(* PLC project marvel_solar, Institute of Astronomy Onto 0.0.1 *)
(* stored: creationDateTime 2025-01-01T00:00:00.0, modificationDateTime 2025-01-01T00:00:00.0 *)

TYPE SolarProcesses : STRUCT
  {attribute 'TcHmiSymbol.Show'}
  initialize : Process;  (* Initialize the solar telescope *)
  {attribute 'TcHmiSymbol.Show'}
  power_on_pc : Process;  (* enable power to to solar pc and mount *)
  {attribute 'TcHmiSymbol.Show'}
  power_off_pc : Process;  (* Stop power to solar pc and mount *)
  {attribute 'TcHmiSymbol.Show'}
  power_on_mount : Process;  (* enable power to to solar mount and mount *)
  {attribute 'TcHmiSymbol.Show'}
  power_off_mount : Process;  (* Stop power to solar mount and mount *)
  {attribute 'TcHmiSymbol.Show'}
  manual_power_on : Process;  (* overwrite hard limits *)
  {attribute 'TcHmiSymbol.Show'}
  manual_power_off : Process;  (* Stop overwriting hard limits *)
END_STRUCT;
END_TYPE

TYPE SolarStatuses : STRUCT
  {attribute 'OPC.UA.DA' := '1'}
  {attribute 'OPC.UA.DA.Access' := '1'}
  {attribute 'TcHmiSymbol.Show'}
  health : HealthStatus;
  {attribute 'OPC.UA.DA' := '1'}
  {attribute 'OPC.UA.DA.Access' := '1'}
  {attribute 'TcHmiSymbol.Show'}
  busy : BusyStatus;  (* True if the solar telescope is busy *)
  {attribute 'OPC.UA.DA' := '1'}
  {attribute 'OPC.UA.DA.Access' := '1'}
  {attribute 'TcHmiSymbol.Show'}
  init : InitializationStatus;  (* True if the solar telescope is initialized *)
END_STRUCT;
END_TYPE

TYPE SolarConfig : STRUCT
  {attribute 'TcHmiSymbol.Show'}
  defPowerFan : LREAL;  (* Power of the cooling fan in percent *)
  {attribute 'TcHmiSymbol.Show'}
  highTemp : LREAL;  (* Fan turned up to max power at this temperature to prevent damage *)
  {attribute 'TcHmiSymbol.Show'}
  maxTemp : LREAL;  (* Maximum allowed temperature before the solar telescope is shut down to prevent damage *)
  {attribute 'TcHmiSymbol.Show'}
  fanEnabled : BOOL;  (* True if the cooling fan is enabled *)
END_STRUCT;
END_TYPE

TYPE M_SM_Solar : STRUCT
  {attribute 'OPC.UA.DA' := '1'}
  {attribute 'OPC.UA.DA.Access' := '1'}
  {attribute 'TcHmiSymbol.Show'}
  temp : REAL;
  {attribute 'OPC.UA.DA' := '1'}
  {attribute 'OPC.UA.DA.Access' := '1'}
  {attribute 'TcHmiSymbol.Show'}
  lsAz1 : BOOL;
  {attribute 'OPC.UA.DA' := '1'}
  {attribute 'OPC.UA.DA.Access' := '1'}
  {attribute 'TcHmiSymbol.Show'}
  lsAz2 : BOOL;
  {attribute 'OPC.UA.DA' := '1'}
  {attribute 'OPC.UA.DA.Access' := '1'}
  {attribute 'TcHmiSymbol.Show'}
  lsAz3 : BOOL;
  {attribute 'OPC.UA.DA' := '1'}
  {attribute 'OPC.UA.DA.Access' := '1'}
  {attribute 'TcHmiSymbol.Show'}
  hsAz : BOOL;
  {attribute 'OPC.UA.DA' := '1'}
  {attribute 'OPC.UA.DA.Access' := '1'}
  {attribute 'TcHmiSymbol.Show'}
  lsAl1 : BOOL;
  {attribute 'OPC.UA.DA' := '1'}
  {attribute 'OPC.UA.DA.Access' := '1'}
  {attribute 'TcHmiSymbol.Show'}
  lsAl2 : BOOL;
  {attribute 'OPC.UA.DA' := '1'}
  {attribute 'OPC.UA.DA.Access' := '1'}
  {attribute 'TcHmiSymbol.Show'}
  hsAl : BOOL;
  {attribute 'OPC.UA.DA' := '1'}
  {attribute 'OPC.UA.DA.Access' := '3'}
  {attribute 'TcHmiSymbol.Show'}
  editableConfig : SolarConfig;
  {attribute 'OPC.UA.DA' := '1'}
  {attribute 'OPC.UA.DA.Access' := '1'}
  {attribute 'TcHmiSymbol.Show'}
  actualStatus : STRING;
  {attribute 'OPC.UA.DA' := '1'}
  {attribute 'OPC.UA.DA.Access' := '1'}
  {attribute 'TcHmiSymbol.Show'}
  config : SolarConfig;
  {attribute 'OPC.UA.DA' := '1'}
  {attribute 'OPC.UA.DA.Access' := '1'}
  {attribute 'TcHmiSymbol.Show'}
  fanOk : BOOL;
  {attribute 'OPC.UA.DA' := '1'}
  {attribute 'OPC.UA.DA.Access' := '1'}
  {attribute 'TcHmiSymbol.Show'}
  powerPC : BOOL;
  {attribute 'OPC.UA.DA' := '1'}
  {attribute 'OPC.UA.DA.Access' := '1'}
  {attribute 'TcHmiSymbol.Show'}
  powerMount : BOOL;
  {attribute 'OPC.UA.DA' := '1'}
  {attribute 'OPC.UA.DA.Access' := '1'}
  {attribute 'TcHmiSymbol.Show'}
  powerFan : REAL;
  {attribute 'OPC.UA.DA' := '1'}
  {attribute 'OPC.UA.DA.Access' := '1'}
  {attribute 'TcHmiSymbol.Show'}
  overwriten : BOOL;
  {attribute 'OPC.UA.DA' := '1'}
  {attribute 'TcHmiSymbol.Show'}
  stat : SolarStatuses;
  {attribute 'OPC.UA.DA' := '1'}
  {attribute 'TcHmiSymbol.Show'}
  proc : M_SM_SolarProcesses;
END_STRUCT;
END_TYPE

TYPE M_SM_SolarProcesses : STRUCT
  {attribute 'TcHmiSymbol.Show'}
  initialize : M_Process;
  {attribute 'TcHmiSymbol.Show'}
  power_on_pc : M_Process;
  {attribute 'TcHmiSymbol.Show'}
  power_off_pc : M_Process;
  {attribute 'TcHmiSymbol.Show'}
  power_on_mount : M_Process;
  {attribute 'TcHmiSymbol.Show'}
  power_off_mount : M_Process;
  {attribute 'TcHmiSymbol.Show'}
  manual_power_on : M_Process;
  {attribute 'TcHmiSymbol.Show'}
  manual_power_off : M_Process;
END_STRUCT;
END_TYPE

FUNCTION_BLOCK SM_Solar
  VAR_INPUT
    {attribute 'OPC.UA.DA' := '1'}
    {attribute 'OPC.UA.DA.Access' := '1'}
    temp AT %I* : REAL;  (* The measured temperature *)
    {attribute 'OPC.UA.DA' := '1'}
    {attribute 'OPC.UA.DA.Access' := '1'}
    lsAz1 : BOOL;  (* limit switch azi 1 (soft) (west) (B1) *)
    {attribute 'OPC.UA.DA' := '1'}
    {attribute 'OPC.UA.DA.Access' := '1'}
    lsAz2 : BOOL;  (* limit switch azi 2 (hard) (nord) (B2) *)
    {attribute 'OPC.UA.DA' := '1'}
    {attribute 'OPC.UA.DA.Access' := '1'}
    lsAz3 : BOOL;  (* limit switch azi 3 (soft) (east) (B3) *)
    {attribute 'OPC.UA.DA' := '1'}
    {attribute 'OPC.UA.DA.Access' := '1'}
    hsAz : BOOL;  (* State of home sensor azi (south) (B4) *)
    {attribute 'OPC.UA.DA' := '1'}
    {attribute 'OPC.UA.DA.Access' := '1'}
    lsAl1 : BOOL;  (* limit switch alti 1 (soft) (top) (B5) *)
    {attribute 'OPC.UA.DA' := '1'}
    {attribute 'OPC.UA.DA.Access' := '1'}
    lsAl2 : BOOL;  (* limit switch alti 2 (hard) (mid) (B6) *)
    {attribute 'OPC.UA.DA' := '1'}
    {attribute 'OPC.UA.DA.Access' := '1'}
    hsAl : BOOL;  (* State of home sensor alti + limit (bottom) (B7) *)
    {attribute 'OPC.UA.DA' := '1'}
    {attribute 'OPC.UA.DA.Access' := '3'}
    editableConfig : SolarConfig;  (* Editable configuration of the solar telescope *)
  END_VAR
  VAR_OUTPUT
    {attribute 'OPC.UA.DA' := '1'}
    {attribute 'OPC.UA.DA.Access' := '1'}
    actualStatus : STRING(50);  (* Current status description *)
    {attribute 'OPC.UA.DA' := '1'}
    {attribute 'OPC.UA.DA.Access' := '1'}
    config : SolarConfig;  (* Configuration of the solar telescope *)
    {attribute 'OPC.UA.DA' := '1'}
    {attribute 'OPC.UA.DA.Access' := '1'}
    fanOk : BOOL;  (* True if the cooling fan is working *)
    {attribute 'OPC.UA.DA' := '1'}
    {attribute 'OPC.UA.DA.Access' := '1'}
    powerPC AT %Q* : BOOL;  (* True if the solar pc is enabled *)
    {attribute 'OPC.UA.DA' := '1'}
    {attribute 'OPC.UA.DA.Access' := '1'}
    powerMount AT %Q* : BOOL;  (* True if the solar mount is enabled *)
    {attribute 'OPC.UA.DA' := '1'}
    {attribute 'OPC.UA.DA.Access' := '1'}
    powerFan AT %Q* : REAL;  (* Power of the cooling fan in percent *)
    {attribute 'OPC.UA.DA' := '1'}
    {attribute 'OPC.UA.DA.Access' := '1'}
    overwriten : BOOL;  (* True if the hard limits are overwritten *)
    {attribute 'OPC.UA.DA' := '1'}
    stat : SolarStatuses;  (* Statuses of the state machine *)
    {attribute 'OPC.UA.DA' := '1'}
    proc : SolarProcesses;  (* Processes of the state machine *)
  END_VAR
  VAR_IN_OUT
    {attribute 'OPC.UA.DA' := '0'}
    activity_ref : ActivityStatus;  (* Shared activity status *)
    {attribute 'OPC.UA.DA' := '0'}
    services_ref : Services;  (* Shared services *)
    {attribute 'OPC.UA.DA' := '0'}
    operator_ref : OperatorStatus;  (* Shared operation status *)
  END_VAR

            proc.initialize();
proc.power_on_pc();
proc.power_off_pc();
proc.power_on_mount( isEnabled := (stat.init = InitializationStatus.initialized) AND ((NOT(powerMount)) AND (NOT(stat.health = HealthStatus.bad))) );
proc.power_off_mount();
proc.manual_power_on();
proc.manual_power_off();

          

METHOD _copyFromModel_SM_Solar
  VAR_IN_OUT
    {attribute 'OPC.UA.DA' := '0'}
    model : M_SM_Solar;
  END_VAR
                  THIS^.editableConfig := model.editableConfig;
THIS^.proc.initialize._copyFromModel_Process( model := model.proc.initialize );
THIS^.proc.power_on_pc._copyFromModel_Process( model := model.proc.power_on_pc );
THIS^.proc.power_off_pc._copyFromModel_Process( model := model.proc.power_off_pc );
THIS^.proc.power_on_mount._copyFromModel_Process( model := model.proc.power_on_mount );
THIS^.proc.power_off_mount._copyFromModel_Process( model := model.proc.power_off_mount );
THIS^.proc.manual_power_on._copyFromModel_Process( model := model.proc.manual_power_on );
THIS^.proc.manual_power_off._copyFromModel_Process( model := model.proc.manual_power_off );

                
END_METHOD

METHOD _copyToModel_SM_Solar
  VAR_IN_OUT
    {attribute 'OPC.UA.DA' := '0'}
    model : M_SM_Solar;
  END_VAR
                  model.temp := THIS^.temp;
model.lsAz1 := THIS^.lsAz1;
model.lsAz2 := THIS^.lsAz2;
model.lsAz3 := THIS^.lsAz3;
model.hsAz := THIS^.hsAz;
model.lsAl1 := THIS^.lsAl1;
model.lsAl2 := THIS^.lsAl2;
model.hsAl := THIS^.hsAl;
model.editableConfig := THIS^.editableConfig;
model.actualStatus := THIS^.actualStatus;
model.config := THIS^.config;
model.fanOk := THIS^.fanOk;
model.powerPC := THIS^.powerPC;
model.powerMount := THIS^.powerMount;
model.powerFan := THIS^.powerFan;
model.overwriten := THIS^.overwriten;
model.stat := THIS^.stat;
THIS^.proc.initialize._copyToModel_Process( model := model.proc.initialize );
THIS^.proc.power_on_pc._copyToModel_Process( model := model.proc.power_on_pc );
THIS^.proc.power_off_pc._copyToModel_Process( model := model.proc.power_off_pc );
THIS^.proc.power_on_mount._copyToModel_Process( model := model.proc.power_on_mount );
THIS^.proc.power_off_mount._copyToModel_Process( model := model.proc.power_off_mount );
THIS^.proc.manual_power_on._copyToModel_Process( model := model.proc.manual_power_on );
THIS^.proc.manual_power_off._copyToModel_Process( model := model.proc.manual_power_off );

                
END_METHOD
END_FUNCTION_BLOCK
